FUNCTION FuzzyOR : real
VAR_INPUT
	ORmethod:eORMethod;
	in1,in2:REAL;
END_VAR

CASE ORmethod OF
	Maximum:
		FuzzyOR:=MAX(in1,in2);
END_CASE

END_FUNCTION

(* stored: Version 1.1.0.1, ProductVersion 3.1.4024.6
   POU FuzzyOR: Id {f4bec6ce-f75c-43f1-92a5-9e043334618a}, SpecialFunc None *)
